// TIA Portal V17 export
// export: Created 2025-03-07T09:19:22.7283635Z, ExportSetting WithDefaults, DisplayName Totally Integrated Automation Portal, DisplayVersion V17 Update 8, DisplayName TIA Portal Openness, DisplayVersion V17 Update 8, DisplayName TIA Portal Version Control Interface, DisplayVersion V17, DisplayName SINAMICS Startdrive Advanced, DisplayVersion V17 SP2, DisplayName SINAMICS Startdrive G110M, G120, G120C, G120D, G120P, G115D, DisplayVersion V17 SP2, DisplayName SINAMICS Startdrive G130, G150, S120, S150, SINAMICS MV, S210, DisplayVersion V17 SP2, DisplayName STEP 7 Professional, DisplayVersion V17 Update 8, DisplayName SINUMERIK ONE STEP 7 Toolbox, DisplayVersion V17 Update 12, DisplayName SINUMERIK 840D sl STEP 7 Toolbox, DisplayVersion V17 Update 12, DisplayName STEP 7 Safety, DisplayVersion V17 Update 6, DisplayName WinCC Advanced, DisplayVersion V17 Update 8
VAR_GLOBAL   // PLC tag table "TAGS_IO_FIXTURES_UNIT_02"
   "/////_UNIT_02_FIXTURES_/////" AT %M4000.0 : Bool;   // /////_UNIT_02_FIXTURES_/////
   "/////_FIXTURE_1_UNIT_02_/////" AT %M4000.1 : Bool;   // /////_FIXTURE_1_UNIT_02_/////
   UNIT_02_FIX_1_GRIPPER_CLOSED_I AT %I1060.4 : Bool;   // UNIT 02 FIXTURE 1 GRIPPER CLOSED INPUT
   UNIT_02_FIX_1_GRIPPER_OPEN_I AT %I1060.5 : Bool;   // UNIT 02 FIXTURE 1 GRIPPER OPEN INPUT
   UNIT_02_FIX_1_CLOSE_GRIPPER_O AT %Q1065.0 : Bool;   // UNIT 02 FIXTURE 1 GRIPPER CLOSE OUTPUT
   UNIT_02_FIX_1_OPEN_GRIPPER_O AT %Q1065.1 : Bool;   // UNIT 02 FIXTURE 1 GRIPPER OPEN OUTPUT
   "/////_FIXTURE_2_UNIT_02_/////" AT %M4000.6 : Bool;   // /////_FIXTURE_2_UNIT_02_/////
   UNIT_02_FIX_2_GRIPPER_CLOSED_I AT %I1060.6 : Bool;   // UNIT 02 FIXTURE 2 GRIPPER CLOSED INPUT
   UNIT_02_FIX_2_GRIPPER_OPEN_I AT %I1060.7 : Bool;   // UNIT 02 FIXTURE 2 GRIPPER OPEN INPUT
   UNIT_02_FIX_2_CLOSE_GRIPPER_O AT %Q1065.2 : Bool;   // UNIT 02 FIXTURE 2 GRIPPER CLOSE OUTPUT
   UNIT_02_FIX_2_OPEN_GRIPPER_O AT %Q1065.3 : Bool;   // UNIT 02 FIXTURE 2 GRIPPER OPEN OUTPUT
   "/////_FIXTURE_3_UNIT_02_/////" AT %M4001.3 : Bool;   // /////_FIXTURE_3_UNIT_02_/////
   UNIT_02_FIX_3_GRIPPER_CLOSED_I AT %I1061.0 : Bool;   // UNIT 02 FIXTURE 3 GRIPPER CLOSED INPUT
   UNIT_02_FIX_3_GRIPPER_OPEN_I AT %I1061.1 : Bool;   // UNIT 02 FIXTURE 3 GRIPPER OPEN INPUT
   UNIT_02_FIX_3_CLOSE_GRIPPER_O AT %Q1065.4 : Bool;   // UNIT 02 FIXTURE 3 GRIPPER CLOSE OUTPUT
   UNIT_02_FIX_3_OPEN_GRIPPER_O AT %Q1065.5 : Bool;   // UNIT 02 FIXTURE 3 GRIPPER OPEN OUTPUT
   "/////_FIXTURE_4_UNIT_02_/////" AT %M4002.0 : Bool;   // /////_FIXTURE_4_UNIT_02_/////
   UNIT_02_FIX_4_GRIPPER_CLOSED_I AT %I1061.2 : Bool;   // UNIT 02 FIXTURE 4 GRIPPER CLOSED INPUT
   UNIT_02_FIX_4_GRIPPER_OPEN_I AT %I1061.3 : Bool;   // UNIT 02 FIXTURE 4 GRIPPER OPEN INPUT
   UNIT_02_FIX_4_CLOSE_GRIPPER_O AT %Q1065.6 : Bool;   // UNIT 02 FIXTURE 4 GRIPPER CLOSE OUTPUT
   UNIT_02_FIX_4_OPEN_GRIPPER_O AT %Q1065.7 : Bool;   // UNIT 02 FIXTURE 4 GRIPPER OPEN OUTPUT
END_VAR
